// TIA Portal project "Tonhaofinal_V13" (V13)

(* hardware
DEVICE "S7300/ET200M station_1"  S7-300 station
   slot 0: "Rail_0"  Rail  6ES7 390-1***0-0AA0
   slot 1: "PS 307 5A_1"  PS 307 5A  6ES7 307-1EA01-0AA0
   slot 2: "PLC_1"  CPU 314C-2 PN/DP  6ES7 314-6EH04-0AB0  V3.3
      slot 2: "PROFINET interface_1"  PN-IO
         slot 1: "Port_1"  Port
         slot 2: "Port_2"  Port
      slot 5: "DI24/DO16_1"  DI24/DO16
      slot 6: "AI5/AO2_1"  AI5/AO2
      slot 7: "Count_1"  Counter
      slot 8: "Positioning_1"  Positioning
   slot 4: "DI32 x 24VDC_1"  DI32 x 24VDC  6ES7 321-1BL00-0AA0
   slot 5: "DO16 x 24VDC / 0.5A_1"  DO16 x 24VDC / 0.5A  6ES7 322-1BH01-0AA0
*)

// ===== PLC "PLC_1"  CPU 314C-2 PN/DP =====

VAR_GLOBAL   // PLC tag table "Default tag table"
   "P0" AT %M0.0 : Bool;
   "P1" AT %M0.1 : Bool;
   "P2" AT %M0.2 : Bool;
   "P3" AT %M0.3 : Bool;
   "P4" AT %M0.4 : Bool;
   "P5" AT %M0.5 : Bool;
   "P6" AT %M0.6 : Bool;
   "P7" AT %M0.7 : Bool;
   "P8" AT %M1.0 : Bool;
   "P9" AT %M1.1 : Bool;
   "t1" AT %M1.2 : Bool;
   "t2" AT %M1.3 : Bool;
   "t3" AT %M1.4 : Bool;
   "t4" AT %M1.5 : Bool;
   "t5" AT %M1.6 : Bool;
   "t6" AT %M1.7 : Bool;
   "t7" AT %M2.0 : Bool;
   "t8" AT %M2.1 : Bool;
   "t9" AT %M2.2 : Bool;
   "t10" AT %M2.3 : Bool;
   "sensor fim esteira" AT %I0.0 : Bool;
   "capacitivo" AT %I0.1 : Bool;
   "Profundidade" AT %I0.2 : Bool;
   "Optico" AT %I0.3 : Bool;
   "Indutivo" AT %I0.4 : Bool;
   "Motor direita" AT %Q4.0 : Bool;
   "Motor esquerda" AT %Q4.1 : Bool;
   "Estende vertical" AT %Q4.2 : Bool;
   "Recua vertical" AT %Q4.3 : Bool;
   "Recua metal" AT %Q4.4 : Bool;
   "Estende metal" AT %Q4.5 : Bool;
   "Recua platico" AT %Q4.6 : Bool;
   "Estende plastico" AT %Q4.7 : Bool;
   "t11" AT %M2.4 : Bool;
   "t12" AT %M2.5 : Bool;
   "P10" AT %M2.6 : Bool;
   "P11" AT %M2.7 : Bool;
   "t0" AT %M3.0 : Bool;
   "Start" AT %I125.4 : Bool;
   "t13" AT %M3.1 : Bool;
   "auto" AT %I125.5 : Bool;
   "relay" AT %Q124.0 : Bool;
   "stop" AT %I125.3 : Bool;
   "stop luz" AT %Q124.5 : Bool;
   "Quit" AT %I125.2 : Bool;
   "quit luz" AT %Q124.6 : Bool;
   "start luz" AT %Q124.4 : Bool;
   "tstop" AT %M3.2 : Bool;
   "pstop" AT %M3.3 : Bool;
   "pquit" AT %M3.4 : Bool;
   "tquit" AT %M3.5 : Bool;
   "pquit2" AT %M3.6 : Bool;
   "tquit2" AT %M3.7 : Bool;
   "tquit3" AT %M4.0 : Bool;
   "pstart" AT %M4.1 : Bool;
   "t14" AT %M4.2 : Bool;
   "t15" AT %M4.3 : Bool;
   "t16" AT %M4.4 : Bool;
   "t17" AT %M4.5 : Bool;
   "t18" AT %M4.6 : Bool;
   "t19" AT %M4.7 : Bool;
   "t20" AT %M5.0 : Bool;
   "p12" AT %M5.1 : Bool;
   "p13" AT %M5.2 : Bool;
   "p14" AT %M5.3 : Bool;
   "p15" AT %M5.4 : Bool;
   "p16" AT %M5.5 : Bool;
   "p17" AT %M5.6 : Bool;
   "p18" AT %M5.7 : Bool;
   "p19" AT %M6.0 : Bool;
   "p20" AT %M6.1 : Bool;
   "p21" AT %M6.2 : Bool;
   "p22" AT %M6.3 : Bool;
   "p23" AT %M6.4 : Bool;
   "p24" AT %M6.5 : Bool;
   "p25" AT %M6.6 : Bool;
   "p26" AT %M6.7 : Bool;
   "p27" AT %M7.0 : Bool;
   "t21" AT %M7.1 : Bool;
   "t22" AT %M7.2 : Bool;
   "t23" AT %M7.3 : Bool;
   "t24" AT %M7.4 : Bool;
   "t25" AT %M7.5 : Bool;
   "t26" AT %M7.6 : Bool;
   "t27" AT %M7.7 : Bool;
   "t28" AT %M8.0 : Bool;
   "t29" AT %M8.1 : Bool;
   "t30" AT %M8.2 : Bool;
   "t31" AT %M8.3 : Bool;
   "t32" AT %M8.4 : Bool;
   "t33" AT %M8.5 : Bool;
   "t34" AT %M8.6 : Bool;
   "t35" AT %M8.7 : Bool;
   "t36" AT %M9.0 : Bool;
   "t37" AT %M9.1 : Bool;
   "t38" AT %M9.2 : Bool;
   "t39" AT %M9.3 : Bool;
   "t40" AT %M9.4 : Bool;
   "t41" AT %M9.5 : Bool;
   "t42" AT %M9.6 : Bool;
   "t43" AT %M9.7 : Bool;
   "p28" AT %M10.0 : Bool;
   "p29" AT %M10.1 : Bool;
   "t44" AT %M10.2 : Bool;
   "t45" AT %M10.3 : Bool;
END_VAR

ORGANIZATION_BLOCK "Main"   // OB1, LAD
TITLE = "Main Program Sweep (Cycle)"
{ S7_Optimized_Access := 'FALSE' }
VERSION : 0.1
   VAR_TEMP
      OB1_EV_CLASS : Byte;   // Bits 0-3 = 1 (Coming event), Bits 4-7 = 1 (Event class 1)
      OB1_SCAN_1 : Byte;   // 1 (Cold restart scan 1 of OB 1), 3 (Scan 2-n of OB 1)
      OB1_PRIORITY : Byte;   // Priority of OB Execution
      OB1_OB_NUMBR : Byte;   // 1 (Organization block 1, OB1)
      OB1_RESERVED_1 : Byte;   // Reserved for system
      OB1_RESERVED_2 : Byte;   // Reserved for system
      OB1_PREV_CYCLE : Int;   // Cycle time of previous OB1 scan (milliseconds)
      OB1_MIN_CYCLE : Int;   // Minimum cycle time of OB1 (milliseconds)
      OB1_MAX_CYCLE : Int;   // Maximum cycle time of OB1 (milliseconds)
      OB1_DATE_TIME : Date_And_Time;   // Date and time OB1 started
   END_VAR
BEGIN
END_ORGANIZATION_BLOCK